Universal Robots PolyScope program: AG_force_demo.urp

Program AG_force_demo (installation=default directory=/programs/AutoGrind createdIn=5.9.1.1031110 lastSavedIn=5.11.11.1010533 robotSerialNumber=20195501059)
Calibrated DH parameters: a=[0.000146, -0.418764, -0.053981, 0.000058, -0.000023, 0]; d=[0.162545, 37.319448, -206.067439, 168.881546, 0.09955, 0.099464]; alpha=[1.57004, -0.001979, 0.002304, 1.570607, -1.57066, 0]; deltaTheta=[0, -0.174616, -1.258233, 1.432844, -0.000001, 0]
BeforeStart
  start_p := get_actual_tcp_pose()
  MoveJ speed 60 deg/s, acceleration 80 deg/s^2 (useActiveTCP=true) feature=Base
    Waypoint Waypoint (Variable): variable=start_p
Robot Program (runOnlyOnce=true)
  MoveL speed 250 mm/s, acceleration 1200 mm/s^2 (useActiveTCP=true) feature=Base
    Waypoint lift: TCP in base x=107.196 y=-507.057 z=163.445 mm, rx=-3.1414 ry=0.0231 rz=0 rad; joints [86.986, -84.905, 107.059, -112.143, -89.967, 177.84] deg; TCP offset x=0 y=0 z=175 mm, rx=0 ry=0 rz=0 rad
    Wait Sleep waitTime=0.5
    Waypoint neutral: TCP in base x=107.21 y=-507.105 z=87.743 mm, rx=3.1415 ry=-0.0231 rz=0 rad; joints [86.983, -79.79, 113.642, -123.846, -89.954, 177.852] deg
  MoveL speed 250 mm/s, acceleration 1200 mm/s^2 (useActiveTCP=true) feature=Base
    MoveDirectionNode (selectedDirection=ZPlus toolParams=0.01, 0.5) feature=Joint_6_name
      Until TOOL_CONTACT_DETECTION (allowActions=false retraction=0.001 decelerationAcceleration=0.5 decelerationAngularAcceleration=34.906585)
  Force Frame feature=Joint_6_name; selection=[0, 0, 1, 0, 0, 0]; wrench=[0, 0, 10, 0, 0, 0]; limitsForce=[0.15, 0.15, 0.15, 1.047198, 1.047198, 1.047198]; limitsMotion=[0.1, 0.1, 0.1, 0.349066, 0.349066, 0.349066]
    Wait Sleep waitTime=0.5
    MoveL speed 10 mm/s, acceleration 1200 mm/s^2 (useActiveTCP=true) feature=Base
      Waypoint plusy (Relative): relativeFromPosition TCP in base x=-0.185 y=-500.839 z=23.866 mm, rx=-0.0034 ry=0.0011 rz=0.0001 rad; joints [74.491, -75.856, 120.68, -135.023, -89.952, 164.527] deg; TCP offset x=0 y=0 z=175 mm, rx=-3.1416 ry=0 rz=0 rad; TCP in base x=-0.166 y=-587.775 z=24.153 mm, rx=-0.0034 ry=0.001 rz=0.0001 rad; joints [76.826, -66.151, 106.294, -130.339, -89.984, 166.851] deg
  MoveL speed 250 mm/s, acceleration 1200 mm/s^2 (useActiveTCP=true) feature=Base
    Waypoint lift: TCP in base x=107.196 y=-507.057 z=163.445 mm, rx=-3.1414 ry=0.0231 rz=0 rad; joints [86.986, -84.905, 107.059, -112.143, -89.967, 177.84] deg; TCP offset x=0 y=0 z=175 mm, rx=0 ry=0 rz=0 rad
    Wait Sleep waitTime=0.5
    Waypoint neutral: TCP in base x=107.21 y=-507.105 z=87.743 mm, rx=3.1415 ry=-0.0231 rz=0 rad; joints [86.983, -79.79, 113.642, -123.846, -89.954, 177.852] deg
  MoveL speed 250 mm/s, acceleration 1200 mm/s^2 (useActiveTCP=true) feature=Base
    MoveDirectionNode (selectedDirection=ZPlus toolParams=0.01, 0.5) feature=Joint_6_name
      Until TOOL_CONTACT_DETECTION (allowActions=false retraction=0.001 decelerationAcceleration=0.5 decelerationAngularAcceleration=34.906585)
  Force Frame feature=Joint_6_name; selection=[0, 0, 1, 0, 0, 0]; wrench=[0, 0, 10, 0, 0, 0]; limitsForce=[0.15, 0.15, 0.15, 1.047198, 1.047198, 1.047198]; limitsMotion=[0.1, 0.1, 0.1, 0.349066, 0.349066, 0.349066]
    Wait Sleep waitTime=0.5
    MoveL speed 10 mm/s, acceleration 1200 mm/s^2 (useActiveTCP=true) feature=Base
      Waypoint plus_rx (Relative): relativeFromPosition TCP in base x=0.017 y=-499.993 z=140.74 mm, rx=0 ry=0 rz=0.0001 rad; joints [74.492, -86.057, 111.945, -115.879, -89.957, 164.503] deg; TCP offset x=0 y=0 z=175 mm, rx=-3.1416 ry=0 rz=0 rad; TCP in base x=0 y=-499.984 z=140.72 mm, rx=0.7093 ry=0 rz=0 rad; joints [78.629, -59.693, 76.97, -67.186, -97.407, 171.344] deg
  MoveL speed 250 mm/s, acceleration 1200 mm/s^2 (useActiveTCP=true) feature=Base
    Waypoint lift: TCP in base x=107.196 y=-507.057 z=163.445 mm, rx=-3.1414 ry=0.0231 rz=0 rad; joints [86.986, -84.905, 107.059, -112.143, -89.967, 177.84] deg; TCP offset x=0 y=0 z=175 mm, rx=0 ry=0 rz=0 rad
